(* IEC 61131-3 sources: Industry-PLC-LLM/data/PLCBEAD_repo/PLCBEAD_PLCEmbed-main/PLC-BEAD/Source/GEB/SQRTN, 1 file *)

(* ---- SQRTN.ST ---- *)
FUNCTION SQRTN:REAL

	VAR_INPUT
		X :	REAL;
		N :	INT;
	END_VAR

	IF N > 0 THEN
		SQRTN := EXP(LN(X) / INT_TO_REAL(n));
	ELSE
		SQRTN := 0.0;
	END_IF;

END_FUNCTION

PROGRAM program0
	VAR
		LocalVar0 : REAL;
		LocalVaR1  : INT;
		LocalOUT  : REAL;
	END_VAR

 	LocalOUT := SQRTN(LocalVar0, LocalVaR1 );

END_PROGRAM
